  SOP710.BoxSensor -> OpcUaClient.SOP710_B1
  SOP711.BoxSensor -> OpcUaClient.SOP711_B1
  SOP712.BoxSensor -> OpcUaClient.SOP712_B1
  SOP714.BoxSensor -> OpcUaClient.SOP714_B1
  SOP715.BoxSensor -> OpcUaClient.SOP715_B1
  SOP716.BoxSensor -> OpcUaClient.SOP716_B1
  SOP717.BoxSensor -> OpcUaClient.SOP717_B1
  SOP723.BoxSensor -> OpcUaClient.SOP723_B1
  SOP722.BoxSensor -> OpcUaClient.SOP722_B1
  SOP721.BoxSensor -> OpcUaClient.SOP721_B1
  SOP713.BoxSensor -> OpcUaClient.SOP713_B1
  OpcUaClient.SOP713_K3 -> SOP713.FrontUp
  OpcUaClient.SOP713_K4 -> SOP713.FrontDown
  OpcUaClient.SOP713_K5 -> SOP713.RearUp
  OpcUaClient.SOP713_K6 -> SOP713.RearDown
  SOP730.BoxSensor -> OpcUaClient.SOP730_B1
  SOP730.FrontDownSensor -> OpcUaClient.SOP730_B2
  SOP730.FrontUpSensor -> OpcUaClient.SOP730_B3
  OpcUaClient.SOP730_K2 -> SOP730.FrontUp
  OpcUaClient.SOP730_K3 -> SOP730.FrontDown
  OpcUaClient.SOP730_K4 -> SOP730.RearUp
  OpcUaClient.SOP730_K5 -> SOP730.RearDown
  OpcUaClient.SOP723_K1 -> Light Curtain Sensor 1.DisableSensor
  OpcUaClient.SOP723_K2 -> Light Curtain Sensor 2.DisableSensor
  OpcUaClient.SOP720_KM4 -> Pallet Dispenser Movement Right.SOP720_KM4
  OpcUaClient.SOP720_KM4 -> Pallet Dispenser Movement Left.SOP720_KM4
  SOP720.PositionSensorB4 -> OpcUaClient.SOP720_B1
  SOP720.PositionSensorB5 -> OpcUaClient.SOP720_B2
  SOP720.PositionSensorB6 -> OpcUaClient.SOP720_B3
  OpcUaClient.SOP720_Pal_Refill -> PalletDispensorMovement.ReFillPallet
  SOP721.ConveyorError -> OpcUaClient.SOP721_FQ1
  SOP721.BoxSensor -> OpcUaClient.SOP721_B1
  SOP722.ConveyorError -> OpcUaClient.SOP722_FQ1
  SOP722.BoxSensor -> OpcUaClient.SOP722_B1
  SOP723.ConveyorError -> OpcUaClient.SOP723_FQ1
  SOP723.BoxSensor -> OpcUaClient.SOP723_B1
  OpcUaClient.SOP721_KM2 -> SOP721.MotorREV
  OpcUaClient.SOP722_KM2 -> SOP722.MotorREV
  OpcUaClient.SOP723_KM2 -> SOP723.MotorREV
  OpcUaClient.SOP721_KM1 -> SOP721.MotorFWD
  OpcUaClient.SOP722_KM1 -> SOP722.MotorFWD
  OpcUaClient.SOP723_KM1 -> SOP723.MotorFWD
  SOP720.PositionSensorB4 -> OpcUaClient.SOP720_B1
  SOP720.PositionSensorB5 -> OpcUaClient.SOP720_B2
  SOP720.PositionSensorB6 -> OpcUaClient.SOP720_B3
  OpcUaClient.SOP720_KM3 -> SOP720.MotorFWD
  OpcUaClient.SOP720_KM4 -> SOP720.MotorREV
  OpcUaClient.SOP720_KM1 -> SOP720.RotateFWD
  OpcUaClient.SOP720_KM2 -> SOP720.RotateREV
  SOP730.BoxSensor -> OpcUaClient.SOP730_B1
  OpcUaClient.SOP730_K2 -> SOP730.FrontUp
  OpcUaClient.SOP730_K3 -> SOP730.FrontDown
  OpcUaClient.SOP730_K4 -> SOP730.RearUp
  OpcUaClient.SOP730_K5 -> SOP730.RearDown
  OpcUaClient.SOP730_KM1 -> SOP730.MotorFWD
  OpcUaClient.SOP730_KM2 -> SOP730.MotorREV
  SOP730.ConveyorError -> OpcUaClient.SOP730_FQ1
  SOP720.ConveyorError -> OpcUaClient.SOP720_FQ1
  OpcUaClient.SOP700_H7 -> SUB700LightBeacon.GreenLight
  OpcUaClient.SOP700_H4 -> SUB700LightBeacon.RedLight
  OpcUaClient.SOP712_KM2 -> SOP712.MotorREV
  OpcUaClient.SOP713_KM2 -> SOP713.MotorREV
  OpcUaClient.SOP714_KM2 -> SOP714.MotorREV
  OpcUaClient.SOP715_KM2 -> SOP715.MotorREV
  OpcUaClient.SOP716_KM2 -> SOP716.MotorREV
  OpcUaClient.SOP717_KM2 -> SOP717.MotorREV
  OpcUaClient.SOP710_KM2 -> SOP710.MotorREV
  OpcUaClient.SOP711_KM2 -> SOP711.MotorREV
  OpcUaClient.SOP720_Pal_Full -> PalletDispensorMovement.Pallet_FilledUp
  OpcUaClient.SOP720_Pal_Dispense -> PalletDispensorMovement.NewPallet
  SOP721.ConveyorError -> OpcUaClient.SOP721_FQ1
  SOP721.BoxSensor -> OpcUaClient.SOP721_B1
  OpcUaClient.SOP721_KM1 -> SOP721.MotorFWD
  OpcUaClient.SOP721_KM2 -> SOP721.MotorREV
  SOP723.BoxSensor -> OP710 Input Product.sensor723
  SOP717.BoxSensor -> OP710 Input Product.sensor717
  SOP717.ConveyorError -> OpcUaClient.SOP717_FQ1
  SOP717.BoxSensor -> OpcUaClient.SOP717_B1
  OpcUaClient.SOP717_KM1 -> SOP717.MotorFWD
  OpcUaClient.SOP717_KM2 -> SOP717.MotorREV
  SOP717.ConveyorError -> OpcUaClient.SOP717_FQ1
  SOP717.BoxSensor -> OpcUaClient.SOP717_B1
  OpcUaClient.SOP717_KM1 -> SOP717.MotorFWD
  OpcUaClient.SOP717_KM2 -> SOP717.MotorREV
  IRB4400_60_196_1.vacuum_on -> OP710 Input Product.VacuumOn_I
  IRB4400_60_196_1.SOP740_ProductPlaced -> OpcUaClient.SOP740_ProductPlaced
  OpcUaClient.SOP740_PickProduct -> IRB4400_60_196_1.SOP740_PickProduct
  SOP717.BoxSensor -> Timer_2.Active
  Timer_2.Output -> IRB4400_60_196_1.new_box
  IRB4400_60_196_1.Create_MB16 -> Timer_2.Reset
  IRB4400_60_196_1.Create_MB16T -> Timer_2.Reset
  IRB4400_60_196_1.Create_MB20 -> Timer_2.Reset
  IRB4400_60_196_1.Create_MB24 -> Timer_2.Reset
  SOP720.PositionSensorB4 -> OpcUaClient.SOP720_B2
  SOP720.PositionSensorB5 -> OpcUaClient.SOP720_B3
  SOP720.PositionSensorB6 -> OpcUaClient.SOP720_B8
  SOP720.ConveyorError -> OpcUaClient.SOP720_FQ1
  SOP720.RotationFeedback -> OpcUaClient.SOP720_FQ2
  OpcUaClient.SOP720_KM3 -> SOP720.MotorFWD
  OpcUaClient.SOP720_KM4 -> SOP720.MotorREV
  OpcUaClient.SOP720_KM1 -> SOP720.RotateFWD
  OpcUaClient.SOP720_KM2 -> SOP720.RotateREV
  SOP723.BoxSensor -> More_Pallets.sensor723
  OpcUaClient.SOP740_Pal_Pos_1 -> IRB4400_60_196_1.Place_First
  OpcUaClient.SOP740_Pal_Pos_2 -> IRB4400_60_196_1.Place_Second
  OpcUaClient.SOP740_Pal_Pos_3 -> IRB4400_60_196_1.Place_Third
  OpcUaClient.SOP700_Faulted -> IRB4400_60_196_1.SOP700_FAULTED
  SOP713.FrontDownSensor -> OpcUaClient.SOP713_B2
  SOP713.RareDownSensor -> OpcUaClient.SOP713_B3
  SOP713.FrontUpSensor -> OpcUaClient.SOP713_B4
  SOP713.RearUpSensor -> OpcUaClient.SOP713_B5
  SOP730.FrontDownSensor -> OpcUaClient.SOP730_B2
  SOP730.RareDownSensor -> OpcUaClient.SOP730_B3
  SOP730.FrontSensor -> OpcUaClient.SOP730_B4
  SOP730.RearSensor -> OpcUaClient.SOP730_B5
  OpcUaClient.Box_MB16T_Acc -> OP710 Input Product.Create_MB16T
  OpcUaClient.Box_MB20_Acc -> OP710 Input Product.Create_MB20
  OpcUaClient.Box_MB24_Acc -> OP710 Input Product.Create_MB24
  OpcUaClient.Box_MB16_Acc -> OP710 Input Product.Create_MB16
  OpcUaClient.Box_MB16_Rej -> OP710 Input Product.Reject_MB16
  OpcUaClient.Box_MB16T_Rej -> OP710 Input Product.Reject_MB16T
  OpcUaClient.Box_MB20_Rej -> OP710 Input Product.Reject_MB20
  OpcUaClient.Box_MB24_Rej -> OP710 Input Product.Reject_MB24
  OP710 Input Product.ProductNr -> OpcUaClient.Box_ProductNr
  OP710 Input Product.IDNumber -> OpcUaClient.Box_IDNumber
  OpcUaClient.Pallet_Creation -> More_Pallets.Create_Pallets
  SOP720.PalletSensor -> OpcUaClient.SOP720_B1
  PalletDispensorMovement.DispensorDown -> OpcUaClient.SOP720_DispensorDown
  PalletDispensorMovement.DispensorMid -> OpcUaClient.SOP720_DispensorMid
  PalletDispensorMovement.DispensorUp -> OpcUaClient.SOP720_DispensorUp
  OpcUaClient.SOP720_KM1 -> SOP720.RotateFWD
  OpcUaClient.SOP720_KM2 -> SOP720.RotateREV
  OpcUaClient.SOP720_KM3 -> SOP720.MotorFWD
  OpcUaClient.SOP720_KM4 -> SOP720.MotorREV
  SOP720.ConveyorError -> OpcUaClient.SOP720_FQ1
  SOP720.PositionSensorB4 -> OpcUaClient.SOP720_B2
  SOP720.PositionSensorB5 -> OpcUaClient.SOP720_B3
  SOP720.PositionSensorB6 -> OpcUaClient.SOP720_B8
  SOP720.Conveyor_Sensor -> OpcUaClient.SOP720_B1
  SOP730.BoxSensor -> IRB4400_60_196_1.Sensor730
  OpcUaClient.SOP723_RetirePallet -> More_Pallets.DeletePallet
  OpcUaClient.SOP720_K5 -> Light Curtain Sensor 4.DisableSensor
  OpcUaClient.SOP720_K6 -> Light Curtain Sensor 3.DisableSensor
  OP710 Input Product.Status -> OpcUaClient.Status
  SOP717.BoxSensor -> OP710 Input Product.sensor717
  OpcUaClient.SOP723_RetirePallet -> OP710 Input Product.RetirePallet
  IRB4400_60_196_1.SOP740_RobotReady -> OpcUaClient.SOP740_RobotReady
  OpcUaClient.SOP740_ProductNr -> IRB4400_60_196_1.ProductNr
  SOP730.FrontSensor -> IRB4400_60_196_1.FrontClampUp730
  OpcUaClient.SOP730_KM1 -> IRB4400_60_196_1.KM1_730
  OpcUaClient.SOP750_K6 -> Door.OpenDoor
  Door.DoorOpened -> OpcUaClient.SOP750_K8
  Door.DoorClosed -> OpcUaClient.SOP750_B2
  Light Curtain Sensor 1.Detection -> OpcUaClient.SOP723_LC1_ON
  Light Curtain Sensor 2.Detection -> OpcUaClient.SOP723_LC2_ON
  Light Curtain Sensor 3.Detection -> OpcUaClient.SOP720_LC2_ON
  Light Curtain Sensor 4.Detection -> OpcUaClient.SOP720_LC1_ON
  OpcUaClient.SOP750_K3 -> IRB4400_60_196_1.ResetSafetyCircuit
  OpcUaClient.SOP720_Pal_DispenseDown -> PalletDispensorMovement.Dispensor_Down
  PalletDispensorMovement.DispensorTop -> OpcUaClient.SOP720_Dispensed

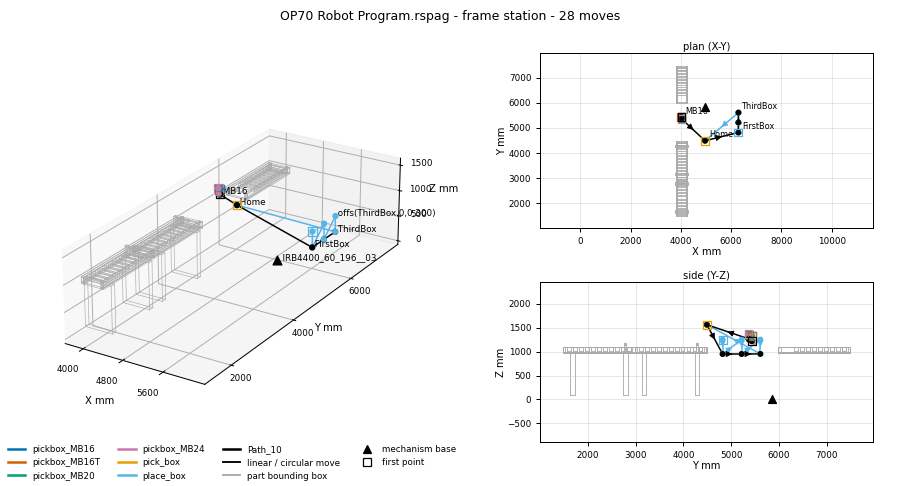
[picture p0: tool path of OP70 Robot Program.rspag in frame station, 28 of 28 moves have a stored position in this frame; points joined in program order, loops and branches not executed]
--- Controller Data/IRB4400_60_196_1/RAPID/TASK1/PROGMOD/CalibData.modx ---
MODULE CalibData
    PERS tooldata vacuum:=[TRUE,[[0,0,175],[1,0,0,0]],[1,[0,0,1],[1,0,0,0],0,0,0]];
ENDMODULE

--- Controller Data/IRB4400_60_196_1/RAPID/TASK1/PROGMOD/MODULE1.modx ---
MODULE MODULE1
    CONST robtarget MB16:=[[418.46,-938.291,1230],[0,0,1,0],[0,0,0,0],[9E+09,9E+09,9E+09,9E+09,9E+09,9E+09]];
    CONST robtarget MB16T:=[[412.744,-943.291,1217.478],[0,0,1,0],[-1,0,-1,0],[9E+09,9E+09,9E+09,9E+09,9E+09,9E+09]];
    CONST robtarget MB20:=[[468.389,-936.264,1247.52],[0,0,1,0],[-1,0,-1,0],[9E+09,9E+09,9E+09,9E+09,9E+09,9E+09]];
    CONST robtarget MB24:=[[482.39,-936.982,1267.685],[0,0,1,0],[-1,0,-1,0],[9E+09,9E+09,9E+09,9E+09,9E+09,9E+09]];
    CONST robtarget Home:=[[1352.798,0,1562.5],[0,0,1,0],[0,0,0,0],[9E+09,9E+09,9E+09,9E+09,9E+09,9E+09]];
    CONST robtarget FirstBox:=[[1024.023,1324.751,949.358],[0,-0.707106781,0.707106781,0],[0,0,0,0],[9E+09,9E+09,9E+09,9E+09,9E+09,9E+09]];
    CONST robtarget SecondBox:=[[626.776,1326.699,949.86],[0,-0.707106781,0.707106781,0],[0,0,0,0],[9E+09,9E+09,9E+09,9E+09,9E+09,9E+09]];
    CONST robtarget ThirdBox:=[[234.737,1327.776,951.145],[0,-0.707106781,0.707106781,0],[0,0,0,0],[9E+09,9E+09,9E+09,9E+09,9E+09,9E+09]];

    VAR intnum interruptEmergency;
    VAR intnum interruptSafety;

    PROC main()

        CONNECT interruptEmergency WITH EmergencyStopTrap;
        ISignalDI SOP700_FAULTED,1,interruptEmergency;

        CONNECT interruptSafety WITH SafetyStopTrap;
        ISignalDI ResetSafetyCircuit,1,interruptSafety;

        setdo SOP740_RobotReady,1;
        WHILE SOP740_RobotReady=1 DO
            IF SOP740_PickProduct=1 THEN
                SetDO SOP740_RobotReady,0;
                pick_box;
                place_box;
            ENDIF
        ENDWHILE
    ENDPROC

    PROC vacuum_activation()
        SetDO vacuum_on,1;
        WaitTime 1;
    ENDPROC

    PROC vacuum_desactivation()
        SetDO vacuum_on,0;
        SetDO SOP740_ProductPlaced,1;
        WaitTime 1;
        SetDO SOP740_ProductPlaced,0;
    ENDPROC

    PROC pickbox_MB16()
        MoveL offs(MB16,0,0,100),v500,fine,vacuum\WObj:=wobj0;
        MoveL MB16,v500,fine,vacuum\WObj:=wobj0;
        vacuum_activation;
        MoveL offs(MB16,0,0,100),v500,fine,vacuum\WObj:=wobj0;
    ENDPROC

    PROC pickbox_MB16T()
        MoveL offs(MB16T,0,0,100),v500,fine,vacuum\WObj:=wobj0;
        MoveL MB16T,v500,fine,vacuum\WObj:=wobj0;
        vacuum_activation;
        MoveL offs(MB16T,0,0,100),v500,fine,vacuum\WObj:=wobj0;
    ENDPROC

    PROC pickbox_MB20()
        MoveL offs(MB20,0,0,100),v500,fine,vacuum\WObj:=wobj0;
        MoveL MB20,v500,fine,vacuum\WObj:=wobj0;
        vacuum_activation;
        MoveL offs(MB20,0,0,100),v500,fine,vacuum\WObj:=wobj0;
    ENDPROC

    PROC pickbox_MB24()
        MoveL offs(MB24,0,0,100),v500,fine,vacuum\WObj:=wobj0;
        MoveL MB24,v500,fine,vacuum\WObj:=wobj0;
        vacuum_activation;
        MoveL offs(MB24,0,0,100),v500,fine,vacuum\WObj:=wobj0;
    ENDPROC

    PROC pick_box()
        pickbox_MB20;
        MoveL Home,v500,z50,vacuum\WObj:=wobj0;
    ENDPROC

    PROC place_box()
        IF Place_First=1 THEN
            MoveL offs(FirstBox,0,0,300),v500,fine,vacuum\WObj:=wobj0;
            WaitDI KM1_730,0;
            WaitDI Sensor730,1;
            WaitDI FrontClampUp730,1;
            MoveL FirstBox,v500,fine,vacuum\WObj:=wobj0;
        ENDIF
        IF Place_Second=1 THEN
            MoveL offs(SecondBox,0,0,300),v500,fine,vacuum\WObj:=wobj0;
            WaitDI KM1_730,0;
            WaitDI Sensor730,1;
            WaitDI FrontClampUp730,1;
            MoveL SecondBox,v500,fine,vacuum\WObj:=wobj0;
        ENDIF
        IF Place_Third=1 THEN
            MoveL offs(ThirdBox,0,0,300),v500,fine,vacuum\WObj:=wobj0;
            WaitDI KM1_730,0;
            WaitDI Sensor730,1;
            WaitDI FrontClampUp730,1;
            MoveL ThirdBox,v500,fine,vacuum\WObj:=wobj0;
        ENDIF
        vacuum_desactivation;
        WaitTime 1;
        MoveL Home,v500,z50,vacuum\WObj:=wobj0;
        SetDO SOP740_RobotReady,1;
        WaitTime 1;
        WaitDI Sensor730, 1;
    ENDPROC


    PROC Path_10()
        MoveL MB16,v1000,z100,vacuum\WObj:=wobj0;
        MoveL MB16T,v1000,z100,vacuum\WObj:=wobj0;
        MoveL MB20,v1000,z100,vacuum\WObj:=wobj0;
        MoveL MB24,v1000,z100,vacuum\WObj:=wobj0;
        MoveL Home,v1000,z100,vacuum\WObj:=wobj0;
        MoveL FirstBox,v1000,z100,vacuum\WObj:=wobj0;
        MoveL SecondBox,v1000,z100,vacuum\WObj:=wobj0;
        MoveL ThirdBox,v1000,z100,vacuum\WObj:=wobj0;
    ENDPROC

    TRAP EmergencyStopTrap
        StopMove;
        TPWrite "Emergency Stop Activated!";
        WaitUntil SOP700_FAULTED=0;
        StartMove;
    ENDTRAP

    TRAP SafetyStopTrap
        StopMove;
        TPWrite "Safety Stop Activated!";
        WaitUntil ResetSafetyCircuit=0;
        StartMove;
    ENDTRAP

    ENDMODULE

--- Controller Data/IRB4400_60_196_1/SYSPAR/EIO.cfg ---
EIO:CFG_1.0:7:0::
#
VIRTUAL_NETWORK:

      -Name "Virtual" -Label "Virtual Device Network"
#
EIO_SIGNAL:

      -Name "Create_MB16" -SignalType "DI"

      -Name "Create_MB16T" -SignalType "DI"

      -Name "Create_MB20" -SignalType "DI"

      -Name "Create_MB24" -SignalType "DI"

      -Name "vacuum_on" -SignalType "DO"

      -Name "ProductNr" -SignalType "GI"

      -Name "SOP700_S1" -SignalType "DO" -Default 1

      -Name "SOP740_RobotReady" -SignalType "DO"

      -Name "SOP740_ProductPlaced" -SignalType "DO"

      -Name "SOP740_PickProduct" -SignalType "DI"

      -Name "Status" -SignalType "DI"

      -Name "Place_First" -SignalType "DI"

      -Name "Place_Second" -SignalType "DI"

      -Name "Place_Third" -SignalType "DI"

      -Name "SOP700_FAULTED" -SignalType "DI"

      -Name "Sensor730" -SignalType "DI"

      -Name "SOP730_Sending" -SignalType "DI"

      -Name "RearDownSensor" -SignalType "DI"

      -Name "FrontClampUp730" -SignalType "DI"

      -Name "KM1_730" -SignalType "DI"

      -Name "ResetSafetyCircuit" -SignalType "DI"

#CTRL_SIGNATURE:VbDr+H0umOkgX77fmcMqyoTzZaFECUdrZp1N+l0Q80Xi3C+4cjX3LsZYgqIGfnhbpiVxwHWXfvSoZiE+imkZDA==

--- Controller Data/IRB4400_60_196_1/SYSPAR/PROC.cfg ---
PROC:CFG_1.0:7:0::

#CTRL_SIGNATURE:Ua5cR5VY5utMJjC/qj5EaxQEt2kKlWU20fE7ci1RXk/3M142IvBR7BaXzhfzURNrm2vA9iIP2vYVbvdnsn/PyA==
